KUKA KRL program: Sps3.sub

&ACCESS RV
&PARAM TPVW_VERSION=8.3.17
DEF  SPS3 ( )
; FOLD ;%{H} %MKUKATPVW
;Init part of vw_usr_s
VW_USR_S (#USR_INIT_SUB3)

LOOP
;Freilaufende SPS
MAKROSUBMIT3()

WAIT FOR NOT $POWER_FAIL
ENDLOOP
END
;ENDFOLD
